FUNCTION FUN_CheckInPos : Bool
VAR_INPUT
	ActPos : LREAL;
	TargetPos:LREAL;
	ToleranceRange : LREAL;
END_VAR
VAR
	MaxPos : LREAL;
	MinPos : LREAL;
END_VAR

MaxPos := TargetPos + ToleranceRange;
MinPos := TargetPos - ToleranceRange;
IF ActPos > MinPos AND ActPos < MaxPos THEN
	FUN_CheckInPos := TRUE;
ELSE
	FUN_CheckInPos := FALSE;
END_IF

END_FUNCTION

(* stored: Version 1.1.0.1, ProductVersion 3.1.4024.13
   POU FUN_CheckInPos: Id {4f8bdb78-9542-4692-8b83-7020767f36a5}, SpecialFunc None *)
